2932:  !Element, Spacer ;
2933:  !Item 101477937 , Rev A ;
2934:  !Last Modified: 2026-01-19 ;
2935:  !Modified by: Aaron ;
2936:  !0.46 IN Height ;
2937:  !3.5 IN ID, 5.8 IN OD, 3.5 Lbs W ;
2938:  !ID Jaw # 1004 ;
2939:  !--------------------------- ;
2940:  IF (R[70]=7937) THEN ;
2941:   ;
2942:  !Define Parameters for INF/OTF ;
2943:  !R[105]=AR[1]=100, 2By3 Sheet ;
2944:  !R[105]=AR[1]=200, 3By4 Sheet ;
2945:  CALL JOB_VAR_SETUP(100) ;
2946:   ;
2947:  !--------------------------- ;
2948:  !Define Parameters for Job ;
2949:  R[1]=1    ;
2950:  R[2]=0    ;
2951:  R[4]=0    ;
2952:  R[67]=20    ;
2953:  !R[85] "INF_JAW_OFFSET"(Hgt) ;
2954:  R[85]=20    ;
2955:  !R[86] "INF_PICK_OFFSET" 50mm/sec ;
2956:  R[86]=2    ;
2957:  !R[87] "MAIN_LOAD_OFFSET" (PRELOA ;
2958:  R[87]=0    ;
2959:  !R[100] "GRIPPER_ID" 3 values ;
2960:  !If =100, ID Grippers Installed ;
2961:  !If =200, OD Grippers Installed ;
2962:  !If =300, OD 45 Degree Grippers ;
2963:  R[100]=100    ;
2964:  !--------------------------- ;
2965:   ;
2966:  !If using previous setup data ;
2967:  IF (R[71]=7937) THEN ;
2968:   ;
2969:  !--------------------------- ;
2970:  !1st: Height of Raw piece ;
2971:  R[190]=31.37    ;
2972:  !2nd: Height of Finish piece ;
2973:  R[191]=25.27    ;
2974:  !3rd: Infeed Height Offset ;
2975:  R[192]=(-268)    ;
2976:  !4th: Outfeed Height Offset ;
2977:  R[193]=(-320)    ;
2978:  !--------------------------- ;
2979:   ;
2980:  CALL CREATE_REG(R[190],R[191],R[192],R[193]) ;
2981:   ;
2982:  ENDIF ;
2983:   ;
2984:  !If new loading or offloading pos ;
2985:  !SET R[104] "IMPORT_LOADPOS" ;
2986:  !SET R[104]=1000, Otherwise NO ;
2987:  R[104]=1000    ;
2988:  IF (R[104]=1000) THEN ;
2989:  !R[260]=43, Preload Pos1 ;
2990:  !R[270]=44, Preload PosFinal ;
2991:  !R[300]=53, Offload PosFinal ;
2992:  !PR[43] Pre-Loading Pos1 ;
2993:  CALL CREATE_PR(43,167.634,(-61.21),332.868,125.606,88.913,123.74) ;
2994:  !PR[44] Final Loading Position ;
2995:  CALL CREATE_PR(44,168.397,(-62.456),330.583,(-139.386),87.88,(-141.147)) ;
2996:  !PR[53] pre-Unloading Position ;
2997:  CALL CREATE_PR(53,(-126.862),94.747,73.49,172.899,(-88.227),(-174.493)) ;
2998:  !PR[54] Final Unloading Position ;
2999:  CALL CREATE_PR(54,(-126.241),95.015,51.542,172.164,(-88.238),(-173.761)) ;
3000:  !PR[56] assitant Unloading preses ;
3001:  CALL CREATE_PR(56,(-133.84),95.467,273.686,(-177.134),(-88.249),175.184) ;
3002:  !PR[57] assitant Unloading preses ;
3003:  CALL CREATE_PR(57,(-135.964),108.085,344.284,(-177.144),(-88.245),175.194) ;
3004:  !PR[58] assitant Unloading preses ;
3005:  CALL CREATE_PR(58,296.854,360.959,378.47,(-91.75),(-.28),88.063) ;
3006:  ENDIF ;
3007:   ;
3008:  !---------------------------- ;
3009:  !SR[1] = "JOB_VAR_ID_GRIP" ;
3010:  !JOB_VAR_COMMON(R[103])'s value ;
3011:  !---------------------------- ;
3012:  !2By3 SR[1] INF, Max 18(Straight) ;
3013:  !R[103]=100 ;
3014:  !2By3 INF 45 Degree Diagonal Shif ;
3015:  !R[103]=110 ;
3016:  !---------------------------- ;
3017:  !3By4 SR[1] INF, Max 36(Straight) ;
3018:  !R[103]=150 ;
3019:  !3By4 INF 45 Degree Diagonal Shif ;
3020:  !R[103]=160 ;
3021:  !---------------------------- ;
3022:  !R[103] "JOB_PROFILE" Selection ;
3023:  R[103]=100    ;
3024:  CALL JOB_VAR_COMMON(R[103]) ;
3025:   ;
3026:  ENDIF ;
3027:   ;
3028:  JMP LBL[9999] ;
3029:   ;
3030:  !Job 101477937 Logic Ends ;
3031:  !--------------------------- ;
3032:   ;
3033:  LBL[8815] ;
3034:  !--------------------------- ;
3035:  !Thimble, Upper ;
3036:  !Item 103058815 , Rev A ;
3037:  !Last Modified: 2026-01-23 ;
3038:  !Modified by: Aaron ;
3039:  !2.0 IN Height ;
3040:  !4.75 IN ID, 5.9 IN OD, 11.0 Lbs ;
3041:  !ID Jaw # 1021 ;
3042:  !--------------------------- ;
3043:  IF (R[70]=8815) THEN ;
3044:   ;
3045:  !Define Parameters for INF/OTF ;
3046:  !R[105]=AR[1]=100, 2By3 Sheet ;
3047:  !R[105]=AR[1]=200, 3By4 Sheet ;
3048:  CALL JOB_VAR_SETUP(100) ;
3049:   ;
3050:  !--------------------------- ;
3051:  !Define Parameters for Job ;
3052:  R[1]=1    ;
3053:  R[2]=0    ;
3054:  R[4]=0    ;
3055:  R[67]=20    ;
3056:  !R[85] "INF_JAW_OFFSET"(Hgt) ;
3057:  R[85]=20    ;
3058:  !R[86] "INF_PICK_OFFSET" 50mm/sec ;
3059:  R[86]=2    ;
3060:  !R[87] "MAIN_LOAD_OFFSET" (PRELOA ;
3061:  R[87]=0    ;
3062:  !R[100] "GRIPPER_ID" 3 values ;
3063:  !If =100, ID Grippers Installed ;
3064:  !If =200, OD Grippers Installed ;
3065:  !If =300, OD 45 Degree Grippers ;
3066:  R[100]=100    ;
3067:  !--------------------------- ;
3068:   ;
3069:  !If using previous setup data ;
3070:  IF (R[71]=8815) THEN ;
3071:   ;
3072:  !--------------------------- ;
3073:  !1st: Height of Raw piece ;
3074:  R[190]=31.37    ;
3075:  !2nd: Height of Finish piece ;
3076:  R[191]=25.27    ;
3077:  !3rd: Infeed Height Offset ;
3078:  R[192]=(-250)    ;
3079:  !4th: Outfeed Height Offset ;
3080:  R[193]=(-320)    ;
3081:  !--------------------------- ;
3082:   ;
3083:  CALL CREATE_REG(R[190],R[191],R[192],R[193]) ;
3084:   ;
3085:  ENDIF ;
3086:   ;
3087:  !If new loading or offloading pos ;
3088:  !SET R[104] "IMPORT_LOADPOS" ;
3089:  !SET R[104]=1000, Otherwise NO ;
3090:  R[104]=1000    ;
3091:  IF (R[104]=1000) THEN ;
3092:  !R[260]=43, Preload Pos1 ;
3093:  !R[270]=44, Preload PosFinal ;
3094:  !R[300]=53, Offload PosFinal ;
3095:  !PR[43] Pre-Loading Pos1 ;
3096:  CALL CREATE_PR(43,167.634,(-61.21),332.868,125.606,88.913,123.74) ;
3097:  !PR[44] Final Loading Position ;
3098:  CALL CREATE_PR(44,168.397,(-62.456),330.583,(-139.386),87.88,(-141.147)) ;
3099:  !PR[53] pre-Unloading Position ;
3100:  CALL CREATE_PR(53,(-126.862),94.747,73.49,172.899,(-88.227),(-174.493)) ;
3101:  !PR[54] Final Unloading Position ;
3102:  CALL CREATE_PR(54,(-126.241),95.015,51.542,172.164,(-88.238),(-173.761)) ;
3103:  !PR[56] assitant Unloading preses ;
3104:  CALL CREATE_PR(56,(-133.84),95.467,273.686,(-177.134),(-88.249),175.184) ;
3105:  !PR[57] assitant Unloading preses ;
3106:  CALL CREATE_PR(57,(-135.964),108.085,344.284,(-177.144),(-88.245),175.194) ;
3107:  !PR[58] assitant Unloading preses ;
3108:  CALL CREATE_PR(58,296.854,360.959,378.47,(-91.75),(-.28),88.063) ;
3109:  ENDIF ;
3110:   ;
3111:  !---------------------------- ;
3112:  !SR[1] = "JOB_VAR_ID_GRIP" ;
3113:  !JOB_VAR_COMMON(R[103])'s value ;
3114:  !---------------------------- ;
3115:  !2By3 SR[1] INF, Max 18(Straight) ;
3116:  !R[103]=100 ;
3117:  !2By3 INF 45 Degree Diagonal Shif ;
3118:  !R[103]=110 ;
3119:  !---------------------------- ;
3120:  !3By4 SR[1] INF, Max 36(Straight) ;
3121:  !R[103]=150 ;
3122:  !3By4 INF 45 Degree Diagonal Shif ;
3123:  !R[103]=160 ;
3124:  !---------------------------- ;
3125:  !R[103] "JOB_PROFILE" Selection ;
3126:  R[103]=100    ;
3127:  CALL JOB_VAR_COMMON(R[103]) ;
3128:   ;
3129:  ENDIF ;
3130:   ;
3131:  JMP LBL[9999] ;
3132:   ;
3133:  !Job 103058815 Logic Ends ;
3134:  !--------------------------- ;
3135:   ;
3136:  LBL[9297] ;
3137:  !--------------------------- ;
3138:  !Housing , Lock ;
3139:  !Item 103209297 , Rev A ;
3140:  !Last Modified: 2026-02-09 ;
3141:  !Modified by: Aaron ;
3142:  !2.20 IN Height ;
3143:  !4.56 IN ID, 5.75 IN OD, 10.0 Lbs ;
3144:  !ID Jaw # 1021 ;
3145:  !--------------------------- ;
3146:  IF (R[70]=9297) THEN ;
3147:   ;
3148:  !Define Parameters for INF/OTF ;
3149:  !R[105]=AR[1]=100, 2By3 Sheet ;
3150:  !R[105]=AR[1]=200, 3By4 Sheet ;
3151:  CALL JOB_VAR_SETUP(100) ;
3152:   ;
3153:  !--------------------------- ;
3154:  !Define Parameters for Job ;
3155:  R[1]=1    ;
3156:  R[2]=1    ;
3157:  R[4]=0    ;
3158:  R[67]=40    ;
3159:  !R[85] "INF_JAW_OFFSET"(Hgt) ;
3160:  R[85]=92.55    ;
3161:  !R[86] "INF_PICK_OFFSET" 50mm/sec ;
3162:  R[86]=0    ;
3163:  !R[87] "MAIN_LOAD_OFFSET" (PRELOA ;
3164:  R[87]=0    ;
3165:  !R[100] "GRIPPER_ID" 3 values ;
3166:  !If =100, ID Grippers Installed ;
3167:  !If =200, OD Grippers Installed ;
3168:  !If =300, OD 45 Degree Grippers ;
3169:  R[100]=100    ;
3170:  !--------------------------- ;
3171:   ;
3172:  !If using previous setup data ;
3173:  IF (R[71]=9297) THEN ;
3174:   ;
3175:  !--------------------------- ;
3176:  !1st: Height of Raw piece ;
3177:  R[190]=62.5    ;
3178:  !2nd: Height of Finish piece ;
3179:  R[191]=55.88    ;
3180:  !3rd: Infeed Height Offset ;
3181:  R[192]=(-280)    ;
3182:  !4th: Outfeed Height Offset ;
3183:  R[193]=(-295)    ;
3184:  !--------------------------- ;
3185:   ;
3186:  CALL CREATE_REG(R[190],R[191],R[192],R[193]) ;
3187:   ;
3188:  ENDIF ;
3189:   ;
3190:  !If new loading or offloading pos ;
3191:  !SET R[104] "IMPORT_LOADPOS" ;
3192:  !SET R[104]=1000, Otherwise NO ;
3193:  R[104]=1000    ;
3194:  IF (R[104]=1000) THEN ;
3195:  !R[260]=43, Preload Pos1 ;
3196:  !R[270]=44, Preload PosFinal ;
3197:  !R[300]=53, Offload PosFinal ;
3198:  !PR[43] Pre-Loading Pos1 ;
3199:  CALL CREATE_PR(43,166.254,(-63.355),291.433,176.598,88.378,174.957) ;
3200:  !PR[44] Final Loading Position ;
3201:  CALL CREATE_PR(44,167.764,(-63.308),345.698,176.636,88.381,175.009) ;
3202:  !PR[53] pre-Unloading Position ;
3203:  CALL CREATE_PR(53,(-124.023),94.789,(-21.116),172.336,(-88.24),(-173.912)) ;
3204:  !PR[54] Final Unloading Position ;
3205:  CALL CREATE_PR(54,(-122.823),94.759,(-60.604),172.448,(-88.24),(-174.018)) ;
3206:  !PR[56] assitant Unloading preses ;
3207:  CALL CREATE_PR(56,(-133.84),95.467,273.686,(-177.134),(-88.249),175.184) ;
3208:  !PR[57] assitant Unloading preses ;
3209:  CALL CREATE_PR(57,(-135.964),108.085,344.284,(-177.144),(-88.245),175.194) ;
3210:  !PR[58] assitant Unloading preses ;
3211:  CALL CREATE_PR(58,296.854,360.959,378.47,(-91.75),(-.28),88.063) ;
3212:  ENDIF ;
3213:   ;
3214:  !---------------------------- ;
3215:  !SR[1] = "JOB_VAR_ID_GRIP" ;
3216:  !JOB_VAR_COMMON(R[103])'s value ;
3217:  !---------------------------- ;
3218:  !2By3 SR[1] INF, Max 18(Straight) ;
3219:  !R[103]=100 ;
3220:  !2By3 INF 45 Degree Diagonal Shif ;
3221:  !R[103]=110 ;
3222:  !---------------------------- ;
3223:  !3By4 SR[1] INF, Max 36(Straight) ;
3224:  !R[103]=150 ;
3225:  !3By4 INF 45 Degree Diagonal Shif ;
3226:  !R[103]=160 ;
3227:  !---------------------------- ;
3228:  !R[103] "JOB_PROFILE" Selection ;
3229:  R[103]=100    ;
3230:  CALL JOB_VAR_COMMON(R[103]) ;
3231:   ;
3232:  ENDIF ;
3233:   ;
3234:  JMP LBL[9999] ;
3235:   ;
3236:  !Job 103209297 Logic Ends ;
3237:  !--------------------------- ;
3238:   ;
3239:  LBL[9394] ;
3240:  !--------------------------- ;
3241:  !Housing, Shear ;
3242:  !Item 102679394 , Rev A ;
3243:  !Last Modified: 2026-04-23 ;
3244:  !Modified by: Aaron ;
3245:  !7.6 IN Height ;
3246:  !3.24 IN ID, 4.5 IN OD, 18.5 Lbs ;
3247:  !ID Jaw # 1013 ;
3248:  !--------------------------- ;
3249:  IF (R[70]=9394) THEN ;
3250:   ;
3251:  !Define Parameters for INF/OTF ;
3252:  !R[105]=AR[1]=100, 2By3 Sheet ;
3253:  !R[105]=AR[1]=200, 3By4 Sheet ;
3254:  CALL JOB_VAR_SETUP(100) ;
3255:   ;
3256:  !--------------------------- ;
3257:  !Define Parameters for Job ;
3258:  R[1]=1    ;
3259:  R[2]=1    ;
3260:  R[4]=1    ;
3261:  R[67]=100    ;
3262:  !R[85] "INF_JAW_OFFSET"(Hgt) ;
3263:  R[85]=165.77    ;
3264:  !R[86] "INF_PICK_OFFSET" 50mm/sec ;
3265:  R[86]=10    ;
3266:  !R[87] "MAIN_LOAD_OFFSET" (PRELOA ;
3267:  R[87]=0    ;
3268:  !R[100] "GRIPPER_ID" 3 values ;
3269:  !If =100, ID Grippers Installed ;
3270:  !If =200, OD Grippers Installed ;
3271:  !If =300, OD 45 Degree Grippers ;
3272:  R[100]=100    ;
3273:  !--------------------------- ;
3274:   ;
3275:  !If using previous setup data ;
3276:  IF (R[71]=9394) THEN ;
3277:   ;
3278:  !--------------------------- ;
3279:  !1st: Height of Raw piece ;
3280:  R[190]=199.6    ;
3281:  !2nd: Height of Finish piece ;
3282:  R[191]=193.039    ;
3283:  !3rd: Infeed Height Offset ;
3284:  R[192]=(-305)    ;
3285:  !4th: Outfeed Height Offset ;
3286:  R[193]=(-170)    ;
3287:  !--------------------------- ;
3288:   ;
3289:  CALL CREATE_REG(R[190],R[191],R[192],R[193]) ;
3290:   ;
3291:  ENDIF ;
3292:   ;
3293:  !If new loading or offloading pos ;
3294:  !SET R[104] "IMPORT_LOADPOS" ;
3295:  !SET R[104]=1000, Otherwise NO ;
3296:  R[104]=1000    ;
3297:  IF (R[104]=1000) THEN ;
3298:  !R[260]=43, Preload Pos1 ;
3299:  !R[270]=44, Preload PosFinal ;
3300:  !R[300]=53, Offload PosFinal ;
3301:  !PR[43] Pre-Loading Pos1 ;
3302:  CALL CREATE_PR(43,162.457,(-62.801),206.813,164.683,88.429,163.365) ;
3303:  !PR[44] Final Loading Position ;
3304:  CALL CREATE_PR(44,164.029,(-63.458),265.803,164.522,88.424,163.194) ;
3305:  !PR[53] pre-Unloading Position ;
3306:  CALL CREATE_PR(53,(-132.356),92.431,275.285,169.998,(-88.273),(-171.223)) ;
3307:  !PR[54] Final Unloading Position ;
3308:  CALL CREATE_PR(54,(-127.733),92.998,120.209,170.139,(-88.272),(-171.355)) ;
3309:  !PR[56] assitant Unloading preses ;
3310:  CALL CREATE_PR(56,(-133.84),95.467,273.686,(-177.134),(-88.249),175.184) ;
3311:  !PR[57] assitant Unloading preses ;
3312:  CALL CREATE_PR(57,(-135.964),108.085,344.284,(-177.144),(-88.245),175.194) ;
3313:  !PR[58] assitant Unloading preses ;
3314:  CALL CREATE_PR(58,296.854,360.959,378.47,(-91.75),(-.28),88.063) ;
3315:  ENDIF ;
3316:   ;
3317:  !---------------------------- ;
3318:  !SR[1] = "JOB_VAR_ID_GRIP" ;
3319:  !JOB_VAR_COMMON(R[103])'s value ;
3320:  !---------------------------- ;
3321:  !2By3 SR[1] INF, Max 18(Straight) ;
3322:  !R[103]=100 ;
3323:  !2By3 INF 45 Degree Diagonal Shif ;
3324:  !R[103]=110 ;
3325:  !---------------------------- ;
3326:  !3By4 SR[1] INF, Max 36(Straight) ;
3327:  !R[103]=150 ;
3328:  !3By4 INF 45 Degree Diagonal Shif ;
3329:  !R[103]=160 ;
3330:  !---------------------------- ;
3331:  !R[103] "JOB_PROFILE" Selection ;
3332:  R[103]=100    ;
3333:  CALL JOB_VAR_COMMON(R[103]) ;
3334:   ;
3335:  ENDIF ;
3336:   ;
3337:  JMP LBL[9999] ;
3338:   ;
3339:  !Job 102679394 Logic Ends ;
3340:  !--------------------------- ;
3341:   ;
3342:  LBL[9654] ;
3343:  !--------------------------- ;
3344:  !ADPTR ;
3345:  !Item 100009654 , Rev B ;
3346:  !Last Modified: 2026-04-02 ;
3347:  !Modified by: Aaron ;
3348:  !6.25 IN Height ;
3349:  !3.16 IN ID, 3.742 IN OD, 25.0 Lb ;
3350:  !ID Jaw # 1007 ;
3351:  !--------------------------- ;
3352:  IF (R[70]=9654) THEN ;
3353:   ;
3354:  !Define Parameters for INF/OTF ;
3355:  !R[105]=AR[1]=100, 2By3 Sheet ;
3356:  !R[105]=AR[1]=200, 3By4 Sheet ;
3357:  CALL JOB_VAR_SETUP(100) ;
3358:   ;
3359:  !--------------------------- ;
3360:  !Define Parameters for Job ;
3361:  R[1]=1    ;
3362:  R[2]=0    ;
3363:  R[4]=0    ;
3364:  R[67]=40    ;
3365:  !R[85] "INF_JAW_OFFSET"(Hgt) ;
3366:  R[85]=105.88    ;
3367:  !R[86] "INF_PICK_OFFSET" 50mm/sec ;
3368:  R[86]=0    ;
3369:  !R[87] "MAIN_LOAD_OFFSET" (PRELOA ;
3370:  R[87]=0    ;
3371:  !R[100] "GRIPPER_ID" 3 values ;
3372:  !If =100, ID Grippers Installed ;
3373:  !If =200, OD Grippers Installed ;
3374:  !If =300, OD 45 Degree Grippers ;
3375:  R[100]=100    ;
3376:  !--------------------------- ;
3377:   ;
3378:  !If using previous setup data ;
3379:  IF (R[71]=9654) THEN ;
3380:   ;
3381:  !--------------------------- ;
3382:  !1st: Height of Raw piece ;
3383:  R[190]=159.28    ;
3384:  !2nd: Height of Finish piece ;
3385:  R[191]=158.75    ;
3386:  !3rd: Infeed Height Offset ;
3387:  R[192]=(-311)    ;
3388:  !4th: Outfeed Height Offset ;
3389:  R[193]=(-235)    ;
3390:  !--------------------------- ;
3391:   ;
3392:  CALL CREATE_REG(R[190],R[191],R[192],R[193]) ;
3393:   ;
3394:  ENDIF ;
3395:   ;
3396:  !If new loading or offloading pos ;
3397:  !SET R[104] "IMPORT_LOADPOS" ;
3398:  !SET R[104]=1000, Otherwise NO ;
3399:  R[104]=1000    ;
3400:  IF (R[104]=1000) THEN ;
3401:  !R[260]=43, Preload Pos1 ;
3402:  !R[270]=44, Preload PosFinal ;
3403:  !R[300]=53, Offload PosFinal ;
3404:  !PR[43] Pre-Loading Pos1 ;
3405:  CALL CREATE_PR(43,165.86,(-61.611),145.429,150.192,89.173,148.558) ;
3406:  !PR[44] Final Loading Position ;
3407:  CALL CREATE_PR(44,167.886,(-62.489),311.377,150.836,89.177,149.22) ;
3408:  !PR[53] pre-Unloading Position ;
3409:  CALL CREATE_PR(53,(-130.481),93.166,172.006,168.789,(-88.281),(-170.136)) ;
3410:  !PR[54] Final Unloading Position ;
3411:  CALL CREATE_PR(54,(-128.735),93.392,117.767,169.08,(-88.268),(-170.429)) ;
3412:  !PR[56] assitant Unloading preses ;
3413:  CALL CREATE_PR(56,(-133.84),95.467,273.686,(-177.134),(-88.249),175.184) ;
3414:  !PR[57] assitant Unloading preses ;
3415:  CALL CREATE_PR(57,(-135.964),108.085,344.284,(-177.144),(-88.245),175.194) ;
3416:  !PR[58] assitant Unloading preses ;
3417:  CALL CREATE_PR(58,296.854,360.959,378.47,(-91.75),(-.28),88.063) ;
3418:  ENDIF ;
3419:   ;
3420:  !---------------------------- ;
3421:  !SR[1] = "JOB_VAR_ID_GRIP" ;
3422:  !JOB_VAR_COMMON(R[103])'s value ;
3423:  !---------------------------- ;
3424:  !2By3 SR[1] INF, Max 18(Straight) ;
3425:  !R[103]=100 ;
3426:  !2By3 INF 45 Degree Diagonal Shif ;
3427:  !R[103]=110 ;
3428:  !---------------------------- ;
3429:  !3By4 SR[1] INF, Max 36(Straight) ;
3430:  !R[103]=150 ;
3431:  !3By4 INF 45 Degree Diagonal Shif ;
3432:  !R[103]=160 ;
3433:  !---------------------------- ;
3434:  !R[103] "JOB_PROFILE" Selection ;
3435:  R[103]=100    ;
3436:  CALL JOB_VAR_COMMON(R[103]) ;
3437:   ;
3438:  ENDIF ;
3439:   ;
3440:  JMP LBL[9999] ;
3441:   ;
3442:  !Job 100009654 Logic Ends ;
3443:  !--------------------------- ;
3444:   ;
3445:  LBL[9990] ;
3446:  !--------------------------- ;
3447:  !KAREL PROGRAM ;
3448:  !Item 1111199990  ;
3449:  !Last Modified: 2026-Sep-17 ;
3450:  !Modified by: Erfan ;
3451:  !--------------------------- ;
3452:  IF (R[70]=9990) THEN ;
3453:   ;
3454:  !Define Parameters for INF/OTF ;
3455:  !R[105]=AR[1]=100, 2By3 Sheet ;
3456:  !R[105]=AR[1]=200, 3By4 Sheet ;
3457:  CALL JOB_VAR_SETUP(100) ;
3458:  CALL GN_CLS_SC_F9 ;
3459:  MESSAGE[ID GRIPPING STARTS] ;
3460:  WAIT 3.00(sec) ;
3461:   ;
3462:  !--------------------------- ;
3463:  !Define Parameters for Job ;
3464:  R[1]=1    ;
3465:  R[2]=0    ;
3466:  R[4]=0    ;
3467:  R[67]=40    ;
3468:  !R[85] "INF_JAW_OFFSET"(Hgt) ;
3469:  R[85]=105.88    ;
3470:  !R[86] "INF_PICK_OFFSET" 50mm/sec ;
3471:  R[86]=0    ;
3472:  !R[87] "MAIN_LOAD_OFFSET" (PRELOA ;
3473:  R[87]=0    ;
3474:  !R[100] "GRIPPER_ID" 3 values ;
3475:  !If =100, ID Grippers Installed ;
3476:  !If =200, OD Grippers Installed ;
3477:  !If =300, OD 45 Degree Grippers ;
3478:  R[100]=100    ;
3479:  !--------------------------- ;
3480:   ;
3481:  !If using previous setup data ;
3482:  IF (R[71]=9990) THEN ;
3483:   ;
3484:  !--------------------------- ;
3485:  !1st: Height of Raw piece ;
3486:  R[190]=159.28    ;
3487:  !2nd: Height of Finish piece ;
3488:  R[191]=158.75    ;
3489:  !3rd: Infeed Height Offset ;
3490:  R[192]=(-311)    ;
3491:  !4th: Outfeed Height Offset ;
3492:  R[193]=(-235)    ;
3493:  !--------------------------- ;
3494:   ;
3495:  CALL CREATE_REG(R[190],R[191],R[192],R[193]) ;
3496:   ;
3497:  ENDIF ;
3498:   ;
3499:  !If new loading or offloading pos ;
3500:  !SET R[104] "IMPORT_LOADPOS" ;
3501:  !SET R[104]=1000, Otherwise NO ;
3502:  R[104]=1000    ;
3503:  IF (R[104]=1000) THEN ;
3504:  !R[260]=43, Preload Pos1 ;
3505:  !R[270]=44, Preload PosFinal ;
3506:  !R[300]=53, Offload PosFinal ;
3507:  !PR[43] Pre-Loading Pos1 ;
3508:  CALL CREATE_PR(43,165.86,(-61.611),145.429,150.192,89.173,148.558) ;
3509:  !PR[44] Final Loading Position ;
3510:  CALL CREATE_PR(44,167.886,(-62.489),311.377,150.836,89.177,149.22) ;
3511:  !PR[53] pre-Unloading Position ;
3512:  CALL CREATE_PR(53,(-130.481),93.166,172.006,168.789,(-88.281),(-170.136)) ;
3513:  !PR[54] Final Unloading Position ;
3514:  CALL CREATE_PR(54,(-128.735),93.392,117.767,169.08,(-88.268),(-170.429)) ;
3515:  !PR[56] assitant Unloading preses ;
3516:  CALL CREATE_PR(56,(-133.84),95.467,273.686,(-177.134),(-88.249),175.184) ;
3517:  !PR[57] assitant Unloading preses ;
3518:  CALL CREATE_PR(57,(-135.964),108.085,344.284,(-177.144),(-88.245),175.194) ;
3519:  !PR[58] assitant Unloading preses ;
3520:  CALL CREATE_PR(58,296.854,360.959,378.47,(-91.75),(-.28),88.063) ;
3521:  ENDIF ;
3522:   ;
3523:  !---------------------------- ;
3524:  !SR[1] = "JOB_VAR_ID_GRIP" ;
3525:  !JOB_VAR_COMMON(R[103])'s value ;
3526:  !---------------------------- ;
3527:  !2By3 SR[1] INF, Max 18(Straight) ;
3528:  !R[103]=100 ;
3529:  !2By3 INF 45 Degree Diagonal Shif ;
3530:  !R[103]=110 ;
3531:  !---------------------------- ;
3532:  !3By4 SR[1] INF, Max 36(Straight) ;
3533:  !R[103]=150 ;
3534:  !3By4 INF 45 Degree Diagonal Shif ;
3535:  !R[103]=160 ;
3536:  !---------------------------- ;
3537:  !R[103] "JOB_PROFILE" Selection ;
3538:  R[103]=100    ;
3539:  CALL JOB_VAR_COMMON(R[103]) ;
3540:   ;
3541:  ENDIF ;
3542:   ;
3543:  JMP LBL[9999] ;
3544:   ;
3545:  !Job 1111199990 Logic Ends ;
3546:  !--------------------------- ;
3547:   ;
3548:  LBL[9999] ;
3549:  END ;
/POS
/END
